{attribute 'GeneratedUsingTerminal: EP7402-0057-0017'}
{attribute addProperty BoxType "EP7402-0057-0017"}
{attribute addProperty Id "A_0055_EP7402_0057_0018EP7402_190E100499"}
{attribute addProperty CRC "811150267"}
{attribute addProperty Size "99"}
TYPE A_0054_EP7402_0057_0017_30592BBB EXTENDS EP7402_190E1004 :
STRUCT
	{attribute addProperty Name "A_0055_EP7402_0057_0018"}
	A_0055_EP7402_0057_0018 : EP7402_190E1004;
END_STRUCT
END_TYPE

(* stored: Version 1.2.0.0, ProductVersion 3.1.4024.9
   DUT A_0054_EP7402_0057_0017_30592BBB: Id {f2ca33b8-0f26-46bc-bb47-ec6aa68e90b0} *)
